PROGRAM MAIN

VAR
	fb_HahaDataStuff : FB_DataStuff;
END_VAR

fb_HahaDataStuff();

END_PROGRAM

(* stored: Version 1.1.0.1, ProductVersion 3.1.4024.12
   POU MAIN: Id {70a99225-3558-42f5-a08a-2dc8467b5de3}, SpecialFunc None *)
